// Mitsubishi GX Works2 project: slave   PLC: FX3U/FX3UC

// global labels: Global1
VAR_GLOBAL
  iSettpunkt_referanse_glob : INT;
  iReferanse_glob : INT;
  bManuell_glob : BOOL;
  bModus_glob : BOOL;
  fManOutput_glob : REAL;
  fRampStep_glob : REAL;
  fSettpunkt_Kp_glob : REAL;
  fSettpunkt_Ki_glob : REAL;
  fSettpunkt_Kd_glob : REAL;
  fKp_glob : REAL;
  fKi_glob : REAL;
  fKd_glob : REAL;
  fTf_glob : REAL;
  fNomPådrag_glob : REAL;
  fKff_glob : REAL;
  bUseI_glob : BOOL;
  bUseD_glob : BOOL;
  fP_glob : REAL;
  fI_glob : REAL;
  fD_glob : REAL;
  fFlow_p_glob : REAL;
  FO_VNT_1 : FO_VNT;
  iFo_glob : INT;
  iVnt_glob AT D1 : INT;
  iFlow_glob : INT;
  fTank_p_glob : REAL;
  fFlowLmin_glob : REAL;
  ALARMSYSTEM_1 : ALARMSYSTEM;
  bResetAlarm_glob : BOOL;
  bAlarmCritLow_glob : BOOL;
  bAlarmLow_glob : BOOL;
  bAlarmHigh_glob : BOOL;
  bAlarmCritHigh_glob : BOOL;
  bEmergency_glob : BOOL;
  bStartAlarm_glob : BOOL;
  bVentil1_glob AT Y004 : BOOL;
  bVentil2_glob AT Y005 : BOOL;
  bVentil3_glob AT Y006 : BOOL;
  AUTOTUNING_1 : AUTOTUNING;
  bStartAuto_glob : BOOL;
  bResetAutotuning_glob : BOOL;
  bAbortAuto_glob : BOOL;
  bFerdigAuto_glob : BOOL;
  fHyst_glob : REAL;
  fKpAuto_glob : REAL;
  fKiAuto_glob : REAL;
  fKdAuto_glob : REAL;
  fTfAuto_glob : REAL;
  ADDA_initiering_1 : ADDA_initiering;
  OPPSTART_1 : OPPSTART;
  FRA_MASTER_1 : FRA_MASTER;
  FRA_TANK_1 : FRA_TANK;
  TIL_MASTER_1 : TIL_MASTER;
  TIL_TANK_1 : TIL_TANK;
  PID_Regulator_1 : PID_Regulator;
  VERDIENDRING_1 : VERDIENDRING;
  iRateSek_glob : INT;
  bForover_glob : BOOL;
  bStart_glob : BOOL;
  bStopp_glob : BOOL;
  bRunning_glob : BOOL;
END_VAR

FUNCTION_BLOCK ADDA_initiering
VAR_INPUT
  input : BOOL;
END_VAR
(* structured ladder/FBD written out as ST: instructions are called as NAME(EN, inputs, outputs); _pN, _eN, _tN stand for wires *)
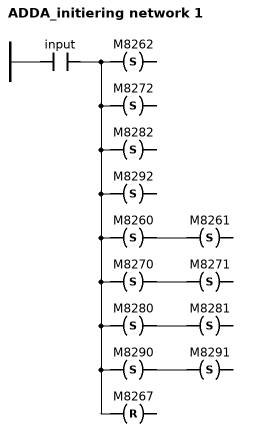
(* network 1 *)
SET(input, M8262);
SET(input, M8272);
SET(input, M8282);
SET(input, M8292);
SET(input, M8260);
SET(input, M8261);
SET(input, M8270);
SET(input, M8271);
SET(input, M8280);
SET(input, M8281);
SET(input, M8290);
SET(input, M8291);
RST(input, M8267);
END_FUNCTION_BLOCK

FUNCTION_BLOCK FO_VNT
VAR_INPUT
  fPID_in : REAL;
  FO : BOOL;
END_VAR
VAR_OUTPUT
  FO_Out : INT;
  VNT_Out : INT;
END_VAR
VAR
  iPID_in : INT;
END_VAR
VAR CONSTANT
  input : BOOL := TRUE;
END_VAR
INT(input,fPID_in,iPID_in);

IF FO THEN
   FO_Out   := REAL_TO_INT(7000.0 + (fPID_in/100.0) * (16384.0 - 7000.0));
   VNT_Out := 4000;
ELSE
   FO_Out   := 16384;
   VNT_Out := iPID_in*45;
END_IF;
END_FUNCTION_BLOCK

FUNCTION_BLOCK Konverter
VAR_INPUT
  rInn : INT;
  maksverdi : INT;
END_VAR
VAR_OUTPUT
  ProsentUt : INT;
END_VAR
VAR_INPUT
  offset : INT;
END_VAR
VAR
  Temp32 : DINT;
END_VAR
Temp32 := INT_TO_DINT(rInn - offset) * 100 / INT_TO_DINT(maksverdi);
ProsentUt:= DINT_TO_INT(Temp32);
END_FUNCTION_BLOCK

FUNCTION_BLOCK PID_Regulator
VAR_INPUT
  referans : INT;
  mea : REAL;
  fKp : REAL;
  fKi : REAL;
  fKd : REAL;
END_VAR
VAR_OUTPUT
  fOut : REAL;
  fP : REAL;
END_VAR
VAR
  fError : REAL;
END_VAR
VAR_OUTPUT
  fI : REAL;
END_VAR
VAR CONSTANT
  fTi : REAL := 10;
  fTs : REAL := 0.01;
END_VAR
VAR_OUTPUT
  fD_term : REAL;
END_VAR
VAR
  fError_prev : REAL;
  fTracking : REAL;
  fNom : REAL;
  bUseI : BOOL;
  bUseD : BOOL;
END_VAR
VAR_INPUT
  fTf : REAL;
END_VAR
VAR CONSTANT
  fTd : REAL := 1.0;
END_VAR
VAR
  fDfilter : REAL;
  fRawOut : REAL;
END_VAR
VAR_INPUT
  fFwd : REAL;
END_VAR
VAR
  bUseFwd : BOOL;
END_VAR
VAR_INPUT
  bMan : BOOL;
END_VAR
VAR
  fKt : REAL;
  fManOutput : REAL;
END_VAR
VAR CONSTANT
  fOutMax : REAL := 100.0;
END_VAR
VAR
  bSaturated : BOOL;
END_VAR
VAR CONSTANT
  fOutMin : REAL;
END_VAR
VAR
  fRef : REAL;
END_VAR
VAR CONSTANT
  input : BOOL := TRUE;
END_VAR
VAR_INPUT
  ManOutput : REAL;
  fKff : REAL;
  bForover : BOOL;
END_VAR
VAR
  bUseI_prev : BOOL;
END_VAR
FLT(input,referans,fRef);

bUseI := fKi > 0.0;
bUseD := fKd > 0.0;

fError:= fRef - mea;

(* P-ledd *)
fP:= fKp*fError;

(* I-ledd *)
IF bUseI THEN
    IF NOT bUseI_prev THEN
        fI := fOut - fP - fD_term - (fFwd * fKff);
    ELSE
        fI := fI + fTs * (fKi * fError + fTracking);
    END_IF;
ELSE
    fI := fNom;
END_IF;
bUseI_prev := bUseI;

(* D-ledd *)
IF bUseD AND fTf > 0.0 THEN
    fDfilter := fDfilter + fTs / fTf * (fKd / fTs * (fError - fError_prev) - fDfilter);
    fD_term := fDfilter;
ELSE
    fD_term := 0.0;
END_IF;

(* foroverkobling *)
fRawOut := fP + fI + fD_term;
IF bForover THEN
    fRawOut := fRawOut + (fFwd * fKff);
END_IF;


IF bMan THEN
    fOut := ManOutput;
    (* Tracking: hold I-ledd oppdatert = rykkfri overgang til auto *)
    fI   := ManOutput - fP- fD_term;
ELSE
    (* Begrens output *)
    IF fRawOut > fOutMax THEN
        fOut    := fOutMax;
        bSaturated := TRUE;
    ELSIF fRawOut < fOutMin THEN
        fOut    := fOutMin;
        bSaturated := TRUE;
    ELSE
        fOut    := fRawOut;
        bSaturated := FALSE;
    END_IF;

    (* Anti-windup tracking signal *)
    fKt := fKi / fKp; (* 1/Ti *)
    fTracking := fKt * (fOut - fRawOut);
END_IF;

 fError_prev:=fError;
END_FUNCTION_BLOCK

PROGRAM PLS_PROGRAM
VAR
  bKlar_glob : BOOL;
END_VAR
(* structured ladder/FBD written out as ST: instructions are called as NAME(EN, inputs, outputs); _pN, _eN, _tN stand for wires *)
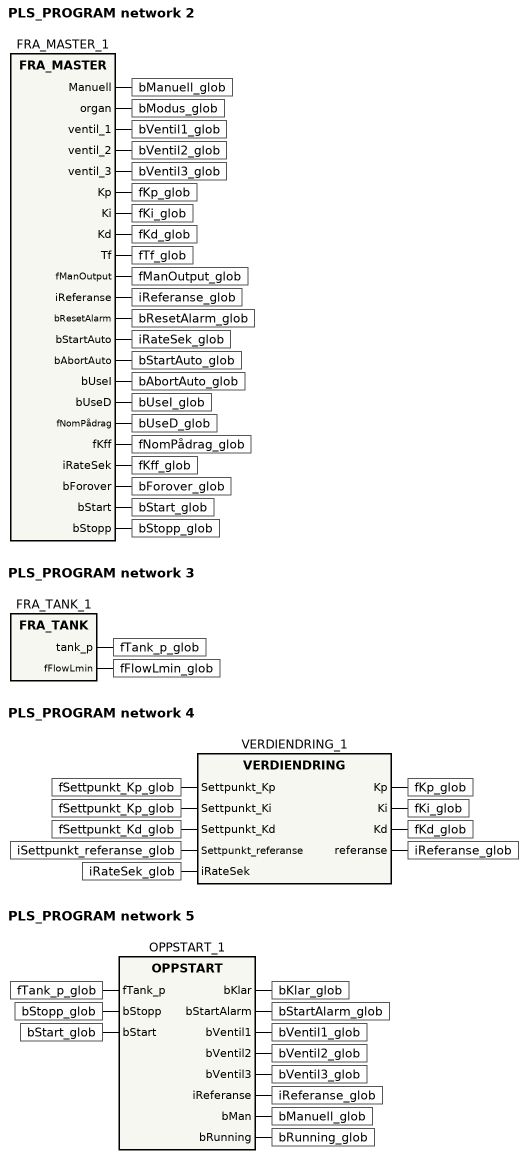
(* network 2 *)
FRA_MASTER_1(Manuell => bManuell_glob, organ => bModus_glob, ventil_1 => bVentil1_glob, ventil_2 => bVentil2_glob, ventil_3 => bVentil3_glob, Kp => fKp_glob, Ki => fKi_glob, Kd => fKd_glob, Tf => fTf_glob, fManOutput => fManOutput_glob, iReferanse => iReferanse_glob, bResetAlarm => bResetAlarm_glob, bStartAuto => iRateSek_glob, bAbortAuto => bStartAuto_glob, bUseI => bAbortAuto_glob, bUseD => bUseI_glob, fNomPådrag => bUseD_glob, fKff => fNomPådrag_glob, iRateSek => fKff_glob, bForover => bForover_glob, bStart => bStart_glob, bStopp => bStopp_glob);
(* network 3 *)
FRA_TANK_1(tank_p => fTank_p_glob, fFlowLmin => fFlowLmin_glob);
(* network 4 *)
VERDIENDRING_1(Settpunkt_Kp := fSettpunkt_Kp_glob, Settpunkt_Ki := fSettpunkt_Kp_glob, Settpunkt_Kd := fSettpunkt_Kd_glob, Settpunkt_referanse := iSettpunkt_referanse_glob, iRateSek := iRateSek_glob, Kp => fKp_glob, Ki => fKi_glob, Kd => fKd_glob, referanse => iReferanse_glob);
(* network 5 *)
OPPSTART_1(fTank_p := fTank_p_glob, bStopp := bStopp_glob, bStart := bStart_glob, bKlar => bKlar_glob, bStartAlarm => bStartAlarm_glob, bVentil1 => bVentil1_glob, bVentil2 => bVentil2_glob, bVentil3 => bVentil3_glob, iReferanse => iReferanse_glob, bMan => bManuell_glob, bRunning => bRunning_glob);
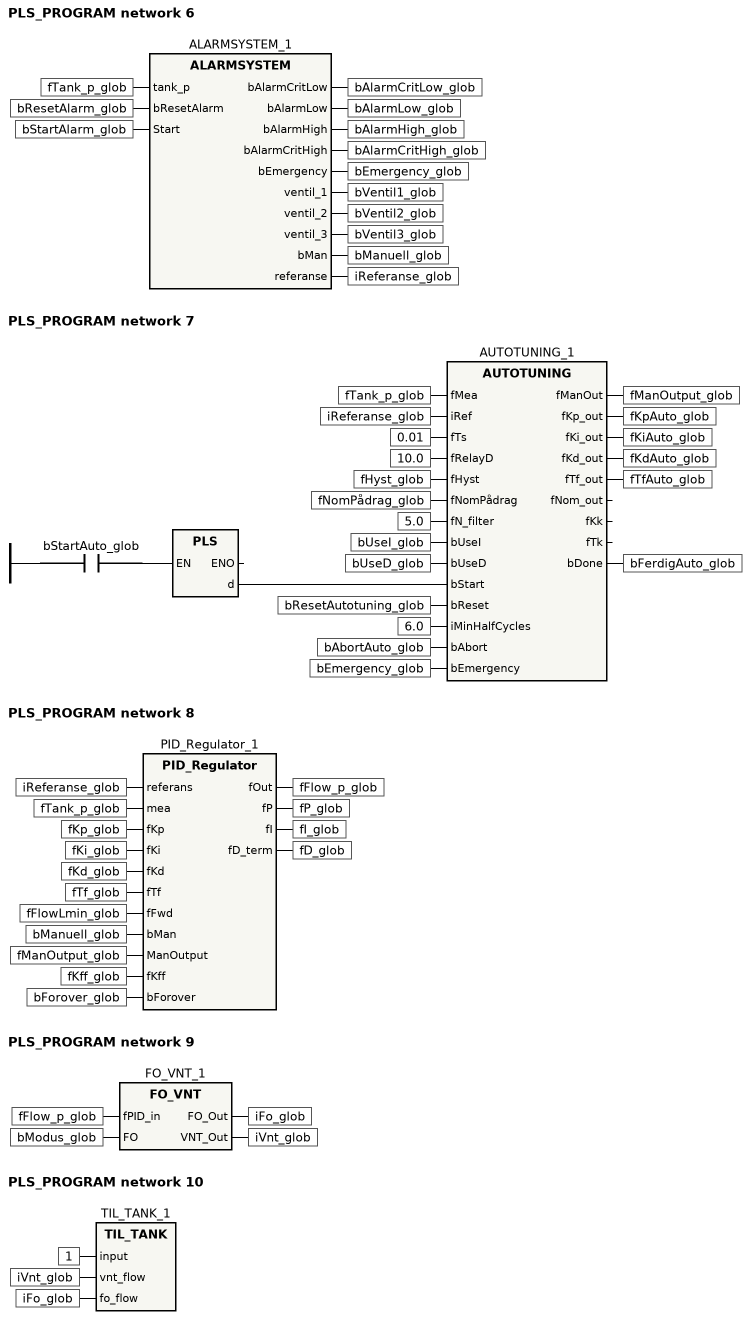
(* network 6 *)
ALARMSYSTEM_1(tank_p := fTank_p_glob, bResetAlarm := bResetAlarm_glob, Start := bStartAlarm_glob, bAlarmCritLow => bAlarmCritLow_glob, bAlarmLow => bAlarmLow_glob, bAlarmHigh => bAlarmHigh_glob, bAlarmCritHigh => bAlarmCritHigh_glob, bEmergency => bEmergency_glob, ventil_1 => bVentil1_glob, ventil_2 => bVentil2_glob, ventil_3 => bVentil3_glob, bMan => bManuell_glob, referanse => iReferanse_glob);
(* network 7 *)
PLS(bStartAuto_glob, _t1);
AUTOTUNING_1(fMea := fTank_p_glob, iRef := iReferanse_glob, fTs := 0.01, fRelayD := 10.0, fHyst := fHyst_glob, fNomPådrag := fNomPådrag_glob, fN_filter := 5.0, bUseI := bUseI_glob, bUseD := bUseD_glob, bStart := _t1, bReset := bResetAutotuning_glob, iMinHalfCycles := 6.0, bAbort := bAbortAuto_glob, bEmergency := bEmergency_glob, fManOut => fManOutput_glob, fKp_out => fKpAuto_glob, fKi_out => fKiAuto_glob, fKd_out => fKdAuto_glob, fTf_out => fTfAuto_glob, bDone => bFerdigAuto_glob);
(* network 8 *)
PID_Regulator_1(referans := iReferanse_glob, mea := fTank_p_glob, fKp := fKp_glob, fKi := fKi_glob, fKd := fKd_glob, fTf := fTf_glob, fFwd := fFlowLmin_glob, bMan := bManuell_glob, ManOutput := fManOutput_glob, fKff := fKff_glob, bForover := bForover_glob, fOut => fFlow_p_glob, fP => fP_glob, fI => fI_glob, fD_term => fD_glob);
(* network 9 *)
FO_VNT_1(fPID_in := fFlow_p_glob, FO := bModus_glob, FO_Out => iFo_glob, VNT_Out => iVnt_glob);
(* network 10 *)
TIL_TANK_1(input := 1, vnt_flow := iVnt_glob, fo_flow := iFo_glob);
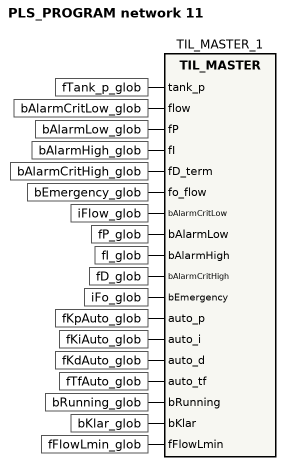
(* network 11 *)
TIL_MASTER_1(tank_p := fTank_p_glob, flow := bAlarmCritLow_glob, fP := bAlarmLow_glob, fI := bAlarmHigh_glob, fD_term := bAlarmCritHigh_glob, fo_flow := bEmergency_glob, bAlarmCritLow := iFlow_glob, bAlarmLow := fP_glob, bAlarmHigh := fI_glob, bAlarmCritHigh := fD_glob, bEmergency := iFo_glob, auto_p := fKpAuto_glob, auto_i := fKiAuto_glob, auto_d := fKdAuto_glob, auto_tf := fTfAuto_glob, bRunning := bRunning_glob, bKlar := bKlar_glob, fFlowLmin := fFlowLmin_glob);
END_PROGRAM

FUNCTION_BLOCK Rampe
VAR_INPUT
  OldValue : REAL;
  NewValue : REAL;
END_VAR
VAR
  RampStep : REAL;
END_VAR
VAR_OUTPUT
  RampOut : REAL;
END_VAR
VAR
  rStartValue : REAL;
  rProgress : REAL;
  rLastTarget : REAL;
  rT_smooth : REAL;
END_VAR
VAR_INPUT
  iRateSek : INT;
END_VAR
VAR
  fRateSek : REAL;
END_VAR
FLT(TRUE, iRateSek, fRateSek);
IF fRateSek < 0.0 THEN
	RampStep := 1.0 / (fRateSek * 100.0);
END_IF;

IF NewValue <> rLastTarget THEN
    rStartValue  := RampOut;
    rProgress    := 0.0;
    rLastTarget  := NewValue;
END_IF;

IF rProgress < 1.0 THEN
    rProgress := rProgress + RampStep;

    IF rProgress > 1.0 THEN
        rProgress := 1.0;
    END_IF;

    (*Smoothstep funksjon, formel: 3t² - 2t³ *)	
    rT_smooth := rProgress * rProgress * (3.0 - (2.0 * rProgress));

    RampOut := rStartValue + ((NewValue - rStartValue) * rT_smooth);
ELSE
    RampOut := NewValue;
END_IF;
END_FUNCTION_BLOCK

FUNCTION_BLOCK TIL_TANK
VAR_INPUT
  input : BOOL;
  vnt_flow : INT;
  fo_flow : INT;
END_VAR
(* structured ladder/FBD written out as ST: instructions are called as NAME(EN, inputs, outputs); _pN, _eN, _tN stand for wires *)
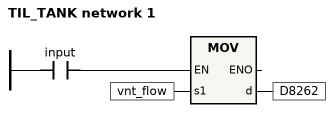
(* network 1 *)
MOV(input, vnt_flow, D8262);
END_FUNCTION_BLOCK

FUNCTION_BLOCK VERDIENDRING
VAR
  Rampe_1 : Rampe;
END_VAR
VAR_INPUT
  Settpunkt_Kp : REAL;
  Settpunkt_Ki : REAL;
  Settpunkt_Kd : REAL;
END_VAR
VAR_OUTPUT
  Kp : REAL;
  Ki : REAL;
  Kd : REAL;
  referanse : INT;
END_VAR
VAR_INPUT
  Settpunkt_referanse : INT;
END_VAR
VAR
  fSettpunkt_referanse : REAL;
  fReferanse : REAL;
  Rampe_2 : Rampe;
  Rampe_3 : Rampe;
  Rampe_4 : Rampe;
END_VAR
VAR_INPUT
  iRateSek : INT;
END_VAR
(* structured ladder/FBD written out as ST: instructions are called as NAME(EN, inputs, outputs); _pN, _eN, _tN stand for wires *)
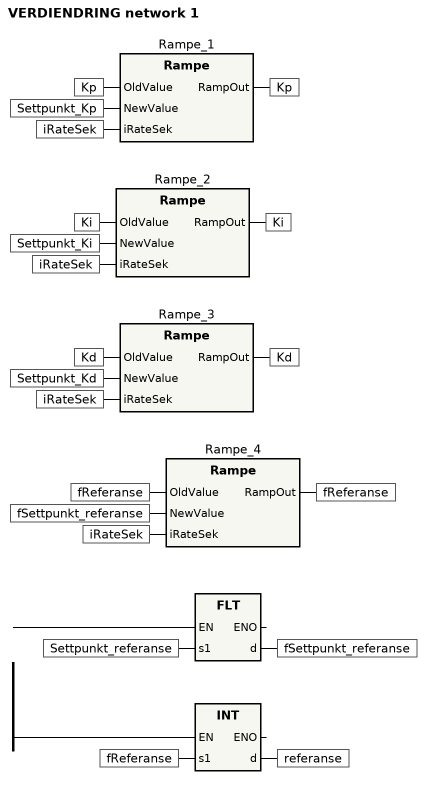
(* network 1 *)
Rampe_1(OldValue := Kp, NewValue := Settpunkt_Kp, iRateSek := iRateSek, RampOut => Kp);
Rampe_2(OldValue := Ki, NewValue := Settpunkt_Ki, iRateSek := iRateSek, RampOut => Ki);
Rampe_3(OldValue := Kd, NewValue := Settpunkt_Kd, iRateSek := iRateSek, RampOut => Kd);
Rampe_4(OldValue := fReferanse, NewValue := fSettpunkt_referanse, iRateSek := iRateSek, RampOut => fReferanse);
FLT(TRUE, Settpunkt_referanse, fSettpunkt_referanse);
INT(TRUE, fReferanse, referanse);
END_FUNCTION_BLOCK

FUNCTION_BLOCK TIL_MASTER
VAR_INPUT
  tank_p : REAL;
  flow : INT;
  fP : REAL;
  fI : REAL;
  fD_term : REAL;
END_VAR
VAR
  iP : INT;
  iI : INT;
  iD : INT;
END_VAR
VAR_INPUT
  fo_flow : INT;
  bAlarmCritLow : BOOL;
  bAlarmLow : BOOL;
  bAlarmHigh : BOOL;
  bAlarmCritHigh : BOOL;
  bEmergency : BOOL;
  auto_p : REAL;
  auto_i : REAL;
  auto_d : REAL;
  auto_tf : REAL;
END_VAR
VAR
  iauto_p : INT;
  iauto_i : INT;
  iauto_d : INT;
  iauto_tf : INT;
  iAlarmWord : INT;
  iStatus : INT;
END_VAR
VAR_INPUT
  bRunning : BOOL;
  bKlar : BOOL;
  fFlowLmin : REAL;
END_VAR
VAR
  iFlowLmin : INT;
END_VAR
(* ===================== TIL MASTER ===================== *)

(* Tank *)
INT(TRUE, tank_p, D23);
TO(TRUE, D23, 0, 10, 1);

(* Pådrag *)
TO(TRUE, flow, 0, 2, 1);

(* Frekvensomformer pådrag *)
TO(TRUE, fo_flow, 0, 3, 1);

(* Pådrag Kp *)
INT(TRUE, fP*1000.0, iP);
TO(TRUE, iP, 0, 4, 1);

(* Pådrag Ki *)
INT(TRUE, fI*1000.0, iI);
TO(TRUE, iI, 0, 5, 1);

(* Pådrag Kd *)
INT(TRUE, fD_term*1000.0, iD);
TO(TRUE, iD, 0, 6, 1);

(* Alarmer *)
iAlarmWord := 0;
IF bAlarmCritLow  THEN iAlarmWord := iAlarmWord + 1;  END_IF;
IF bAlarmLow      THEN iAlarmWord := iAlarmWord + 2;  END_IF; 
IF bAlarmCritHigh THEN iAlarmWord := iAlarmWord + 4;  END_IF;  
IF bAlarmHigh     THEN iAlarmWord := iAlarmWord + 8;  END_IF; 
IF bEmergency     THEN iAlarmWord := iAlarmWord + 16; END_IF; 
TO(TRUE, iAlarmWord, 0, 7, 1);

(* Autotuning *)
IF bFerdigAuto_glob THEN
	INT(TRUE, auto_p*1000.0, iauto_p);
	TO(TRUE, iauto_p, 0, 11, 1);
	
	INT(TRUE, auto_i*1000.0, iauto_i);
	TO(TRUE, iauto_i, 0, 12, 1);
	
	INT(TRUE,auto_d*1000.0, iauto_d);
	TO(TRUE, iauto_d, 0, 13, 1);
	
	INT(TRUE,auto_tf*1000.0, iauto_tf);
	TO(TRUE, iauto_tf, 0, 14, 1);
END_IF;

(* Oppstart *)

iStatus := 0;
IF bRunning AND NOT bKlar THEN iStatus := 1; END_IF;
IF bRunning AND bKlar    THEN iStatus := 2; END_IF; 

TO(TRUE, iStatus, 0, 15, 1);

(* Utstrømsmåling *)
INT(TRUE, fFlowLmin*1000.0, iFlowLmin);
TO(TRUE, iFlowLmin, 0, 1, 1);
END_FUNCTION_BLOCK

FUNCTION_BLOCK ALARMSYSTEM
VAR_INPUT
  tank_p : REAL;
END_VAR
VAR_OUTPUT
  bAlarmCritLow : BOOL;
  bAlarmLow : BOOL;
  bAlarmHigh : BOOL;
  bAlarmCritHigh : BOOL;
  bEmergency : BOOL;
  ventil_1 : BOOL;
  ventil_2 : BOOL;
  ventil_3 : BOOL;
  bMan : BOOL;
  referanse : INT;
END_VAR
VAR_INPUT
  bResetAlarm : BOOL;
END_VAR
VAR
  timer : BOOL;
END_VAR
VAR_INPUT
  Start : BOOL;
END_VAR
VAR CONSTANT
  fSafeKp : REAL := 1.2;
  fSafeKi : REAL := 0.1;
  fSafeKd : REAL := 0.8;
END_VAR
IF Start THEN
    bAlarmCritLow  := tank_p < 10.0;
    bAlarmLow      := tank_p < 20.0 AND NOT bAlarmCritLow;
    bAlarmHigh     := tank_p > 80.0 AND NOT bAlarmCritHigh;
    bAlarmCritHigh := tank_p > 90.0;

    IF bAlarmCritHigh OR bAlarmCritLow THEN
        bEmergency := TRUE;
        fKp_glob := fSafeKp;
        fKi_glob := fSafeKi;
        fKd_glob := fSafeKd;
        ventil_1 := TRUE;
        ventil_2 := TRUE;
        ventil_3 := FALSE;
        referanse := 50;
        bMan := FALSE;
    END_IF;

    IF bEmergency THEN
        ventil_1 := TRUE;
        ventil_2 := TRUE;
        ventil_3 := FALSE;
        referanse := 50;
        bMan := FALSE;

        IF tank_p > 45.0 AND tank_p < 55.0 THEN
            timer := TRUE;
            OUT_T(timer, TC0, 50);
            IF TS0 THEN
                bMan := TRUE;
                fManOutput_glob := 0.0;
                ventil_1 := FALSE;
                ventil_2 := FALSE;
                ventil_3 := FALSE;
            END_IF;
        ELSE
            timer := FALSE;
        END_IF;

        IF bResetAlarm AND tank_p > 45.0 AND tank_p < 55.0 THEN
            bEmergency     := FALSE;
            bAlarmCritLow  := FALSE;
            bAlarmCritHigh := FALSE;
            ventil_1 := TRUE;
            ventil_2 := TRUE;
            ventil_3 := FALSE;
        END_IF;
    END_IF;
END_IF;
END_FUNCTION_BLOCK

FUNCTION_BLOCK FRA_MASTER
VAR_OUTPUT
  Manuell : BOOL;
  organ : BOOL;
  ventil_1 : BOOL;
  ventil_2 : BOOL;
  ventil_3 : BOOL;
  Kp : REAL;
  Ki : REAL;
  Kd : REAL;
  Tf : REAL;
  fManOutput : REAL;
  iReferanse : INT;
  bResetAlarm : BOOL;
  bStartAuto : BOOL;
  bAbortAuto : BOOL;
  bUseI : BOOL;
  bUseD : BOOL;
  fNomPådrag : REAL;
  fKff : REAL;
  iRateSek : INT;
  bForover : BOOL;
  bStart : BOOL;
  bStopp : BOOL;
END_VAR
(* ===================== FRA MASTER ===================== *)

(*  Referanse *)
FROM(TRUE, 0, 0, 1, D10);

IF iReferanse<> D10 THEN
    iReferanse:= D10;
END_IF;

(* Ventiler *)
FROM(TRUE, 0, 1, 1, D11);
ventil_1   := D11.0;
ventil_2   := D11.1;
ventil_3   := D11.2;

(* PID-parametere*)

(* Kp *)
FROM(TRUE, 0, 4, 1, D14);
FLT(TRUE, D14, Kp);
Kp := Kp/1000.0;

(* Ki *)
FROM(TRUE, 0, 5, 1, D16);
FLT(TRUE, D16, Ki);
Ki := Ki/1000.0;

(* Kd *)
FROM(TRUE, 0, 6, 1, D18);
FLT(TRUE, D18, Kd);
Kd := Kd/1000.0;

(* Tf *)
FROM(TRUE, 0, 8, 1, D20);
FLT(TRUE, D20, Tf);
Tf := Tf/1000.0;

(* Manuelt pådrag *)
FROM(TRUE, 0, 9, 1, D22);
FLT(TRUE, D22, fManOutput);
fManOutput := fManOutput/100.0;

(* Organ *)
Organ      := D11.3;

(* manuell eller auto *)
Manuell    := D11.4;

(* Reset alarm *)
bResetAlarm := D11.5;

(* Bruk foroverkobling *)
bForover := D11.6;

(* Start/stopp *)
bStart := D11.7;
bStopp := D11.8;

(* Autotuning *)
FROM(TRUE, 0, 12, 1, D28);

bStartAuto  := D28.0;
bAbortAuto := D28.4;

IF D28.2 THEN
    bUseI := TRUE;
ELSE
    bUseI := FALSE;
END_IF;

IF D28.3 THEN
    bUseD := TRUE;
ELSE
    bUseD := FALSE;
END_IF;


(* Nom pådrag *)
FROM(TRUE, 0, 13, 1, D29);
FLT(TRUE, D29, fNomPådrag);
fNomPådrag := fNomPådrag/100.0;

(* Foroverkoblingskoeffisient *)
FROM(TRUE, 0, 14, 1, D30);
FLT(TRUE, D30, fKff);
fKff:= fKff/100.0;

(* Ratebegrensning *)
FROM(TRUE, 0, 15, 1, D31);
iRateSek := D31;
END_FUNCTION_BLOCK

FUNCTION_BLOCK FRA_TANK
VAR
  fAlpha : REAL;
  tank_p_raw : REAL;
  tank_p_filt : REAL;
  bFirstRun : BOOL;
END_VAR
VAR_OUTPUT
  tank_p : REAL;
END_VAR
VAR
  tank : INT;
  ftank : REAL;
  fFlow_raw : REAL;
END_VAR
VAR_OUTPUT
  fFlowLmin : REAL;
END_VAR
(* Tank i råverdi *)
MOV(TRUE, D8260, tank);

(* Tank i prosent *)
FLT(TRUE, tank, ftank);
tank_p_raw := ((ftank - 500.0) * 100.0) / (1550.0 - 500.0);

fAlpha := 0.02;
IF NOT bFirstRun THEN
    tank_p_filt := tank_p_raw;
    bFirstRun := TRUE;
ELSE
    tank_p_filt := fAlpha * tank_p_raw + (1.0 - fAlpha) * tank_p_filt;
END_IF;
tank_p := tank_p_filt;


(* Strømningsmåler *)
FLT(TRUE,D8261, fFlow_raw);
fFlowLmin := ((fFlow_raw - 400.0) / (1800.0 - 400.0)) * 6.6;
IF fFlowLmin < 0.0 THEN fFlowLmin := 0.0; END_IF;
END_FUNCTION_BLOCK

FUNCTION_BLOCK AUTOTUNING
VAR_INPUT
  fMea : REAL;
  iRef : INT;
  fTs : REAL;
  fRelayD : REAL;
  fHyst : REAL;
  fNomPådrag : REAL;
  fN_filter : REAL;
  bUseI : BOOL;
  bUseD : BOOL;
  bStart : BOOL;
  bReset : BOOL;
  iMinHalfCycles : REAL;
END_VAR
VAR_OUTPUT
  fManOut : REAL;
  fKp_out : REAL;
  fKi_out : REAL;
  fKd_out : REAL;
  fTf_out : REAL;
  fNom_out : REAL;
  fKk : REAL;
  fTk : REAL;
  bDone : BOOL;
END_VAR
VAR
  fError : REAL;
  fError_prev : REAL;
  fPeakHigh : REAL;
  fPeakLow : REAL;
  fAmplitude : REAL;
  fPeriod : REAL;
  fLastCrossTime : REAL;
  fCycleTimer : REAL;
  iHalfCycles : REAL;
  bRelayState : BOOL;
  bInitDone : BOOL;
  fTd_temp : REAL;
  bRunning : BOOL;
  fRef : REAL;
END_VAR
VAR_INPUT
  bAbort : BOOL;
  bEmergency : BOOL;
END_VAR
VAR
  bStartLatch : BOOL;
  fMeaFilt : REAL;
  bWasManual : BOOL;
END_VAR
FLT(TRUE, iRef, fRef);

(* Reset *)
IF bReset THEN
    fError         := 0.0;
    fError_prev    := 0.0;
    fPeakHigh      := -1.0E+30;
    fPeakLow       := 1.0E+30;
    fAmplitude     := 0.0;
    fPeriod        := 0.0;
    fLastCrossTime := 0.0;
    fCycleTimer    := 0.0;
    iHalfCycles    := 0.0;
    bRelayState    := FALSE;
    bInitDone      := FALSE;
    bRunning       := FALSE;
    bDone          := FALSE;
    fManOut        := fNomPådrag;
    fKp_out        := 0.0;
    fKi_out        := 0.0;
    fKd_out        := 0.0;
    fTf_out        := 0.0;
    fNom_out       := 0.0;
    fKk        := 0.0;
    fTk        := 0.0;
    RETURN;
END_IF;

(* Latch start-puls *)
IF bStart THEN
    bStartLatch := TRUE;
END_IF;

(* Start-flanke: initialiser *)
IF bStartLatch AND (NOT bInitDone) AND (NOT bDone) THEN
    bWasManual     := bManuell_glob;

    fPeakHigh      := -1.0E+30;
    fPeakLow       := 1.0E+30;
    fCycleTimer    := 0.0;
    fLastCrossTime := 0.0;
    iHalfCycles    := 0.0;
    fError_prev    := 0.0;
    bRelayState    := FALSE;
    bRunning       := TRUE;
    bDone          := FALSE;
    bInitDone      := TRUE;
    fManOut        := fNomPådrag;
    bStartLatch    := FALSE;
END_IF;

(* Hoveddel *)
IF bRunning THEN

    bManuell_glob   := TRUE;
    fManOutput_glob := fManOut;

    IF bAbort OR bEmergency THEN
        bRunning      := FALSE;
        bDone         := FALSE;
        bInitDone     := FALSE;
        bManuell_glob := bWasManual;
        fManOut       := fNomPådrag;
        RETURN;
    END_IF;

    fError := fRef - fMea;
    fCycleTimer := fCycleTimer + fTs;

    IF fError > fHyst THEN
        bRelayState := TRUE;
    ELSIF fError < -fHyst THEN
        bRelayState := FALSE;
    END_IF;

    IF bRelayState THEN
        fManOut := fNomPådrag + fRelayD;
    ELSE
        fManOut := fNomPådrag - fRelayD;
    END_IF;

    IF (fError * fError_prev < 0.0) THEN

        IF iHalfCycles >= iMinHalfCycles THEN
            fAmplitude := (fPeakHigh - fPeakLow) / 2.0;

            IF fAmplitude > 0.0 THEN
                (* Kritisk forsterkning og kritisk periodetid *)
                fKk := (4.0 * fRelayD) / (3.14159 * fAmplitude);
                fTk := fPeriod;

                (* P *)
                IF (NOT bUseI) AND (NOT bUseD) THEN
                    fKp_out  := 0.5 * fKk;
                    fKi_out  := 0.0;
                    fKd_out  := 0.0;
                    fTf_out  := 0.0;
                    fNom_out := fNomPådrag;

                (* PI — Tyreus-Luyben *)
                ELSIF bUseI AND (NOT bUseD) THEN
                    fKp_out  := fKk / 3.2;
                    fKi_out  := fKp_out / (2.2 * fTk);
                    fKd_out  := 0.0;
                    fTf_out  := 0.0;
                    fNom_out := 0.0;

                (* PD *)
                ELSIF (NOT bUseI) AND bUseD THEN
                    fKp_out  := 0.5 * fKk;
                    fKi_out  := 0.0;
                    fTd_temp := fTk / 8.0;
                    fKd_out  := fKp_out * fTd_temp;
                    fNom_out := fNomPådrag;
                    IF fN_filter > 0.0 THEN
                        fTf_out := fTd_temp / fN_filter;
                    ELSE
                        fTf_out := 0.0;
                    END_IF;

                (* PID — Tyreus-Luyben *)
                ELSIF bUseI AND bUseD THEN
                    fKp_out  := fKk / 3.2;
                    fKi_out  := fKp_out / (2.2 * fTk);
                    fTd_temp := fTk/ 6.3;
                    fKd_out  := fKp_out * fTd_temp;
                    fNom_out := 0.0;
                    IF fN_filter > 0.0 THEN
                        fTf_out := fTd_temp / fN_filter;
                    ELSE
                        fTf_out := 0.0;
                    END_IF;
                END_IF;
            END_IF;

            bDone           := TRUE;
            bRunning        := FALSE;
            bManuell_glob   := bWasManual;
            fManOutput_glob := fNomPådrag;
            fManOut         := fNomPådrag;
        END_IF;

        IF iHalfCycles > 0.0 THEN
            fPeriod := 2.0 * (fCycleTimer - fLastCrossTime);
        END_IF;
        fLastCrossTime := fCycleTimer;
        iHalfCycles := iHalfCycles + 1.0;

        fPeakHigh := -1.0E+30;
        fPeakLow  := 1.0E+30;
    END_IF;

    IF fMea > fPeakHigh THEN fPeakHigh := fMea; END_IF;
    IF fMea < fPeakLow  THEN fPeakLow  := fMea; END_IF;

    fError_prev := fError;
END_IF;
END_FUNCTION_BLOCK

FUNCTION_BLOCK OPPSTART
VAR_OUTPUT
  bKlar : BOOL;
  bStartAlarm : BOOL;
  bVentil1 : BOOL;
  bVentil2 : BOOL;
  bVentil3 : BOOL;
  iReferanse : INT;
  bMan : BOOL;
END_VAR
VAR_INPUT
  fTank_p : REAL;
END_VAR
VAR
  bStartupTimer : BOOL;
END_VAR
VAR_OUTPUT
  bRunning : BOOL;
END_VAR
VAR_INPUT
  bStopp : BOOL;
  bStart : BOOL;
END_VAR
IF bStopp THEN
    bKlar := FALSE;
    bRunning := FALSE;
    bStartAlarm := FALSE;
    bVentil1 := FALSE;
    bVentil2 := FALSE;
    bVentil3 := FALSE;
    bMan := TRUE;
    fManOutput_glob := 0.0;
    bStartupTimer := FALSE;
    RETURN;
END_IF;

IF bStart AND NOT bRunning THEN
    bRunning := TRUE;
    bKlar := FALSE;
END_IF;

IF bRunning THEN
    IF NOT bKlar THEN
        bStartAlarm := FALSE;
        bVentil1 := TRUE;
        bVentil2 := TRUE;
        bVentil3 := FALSE;
        iReferanse := 50;
        bMan := FALSE;
        IF fTank_p > 40.0 AND fTank_p < 60.0 THEN
            bStartupTimer := TRUE;
            OUT_T(bStartupTimer, TC1, 50);
            IF TS1 THEN
                bKlar := TRUE;
                bStartAlarm := TRUE;
            END_IF;
        ELSE
            bStartupTimer := FALSE;
        END_IF;
    ELSE
        bStartAlarm := TRUE;
    END_IF;
END_IF;
END_FUNCTION_BLOCK
